PROGRAM MAIN
VAR
	k :INT;
	
	s1 : DUT1;
	s2 : DUT2;
END_VAR

s1.b := TRUE;
s1.i := 99;
s1.j := 9.9;

s2 := s1;

END_PROGRAM

(* stored: Version 1.1.0.1, ProductVersion 3.1.4024.12
   POU MAIN: Id {be47a598-5e55-462e-87a5-ac47a191ec4d}, SpecialFunc None *)
